TYPE ST_Steuerung_auto_manu_opti_AMPELSIGNAL :
STRUCT
	auto			: ST_System_Ampel_Signal;
	manu			: ST_System_Ampel_Signal;
	manu_Modus		: BOOL;
	opti			: ST_System_Ampel_Signal;
	opti_Modus		: BOOL;
END_STRUCT
END_TYPE

(* stored: Version 1.1.0.1, ProductVersion 3.1.4024.9
   DUT ST_Steuerung_auto_manu_opti_AMPELSIGNAL: Id {8e408c61-0068-41de-b554-1980eebc63fb} *)
